RoboDK station: ur3.rdk

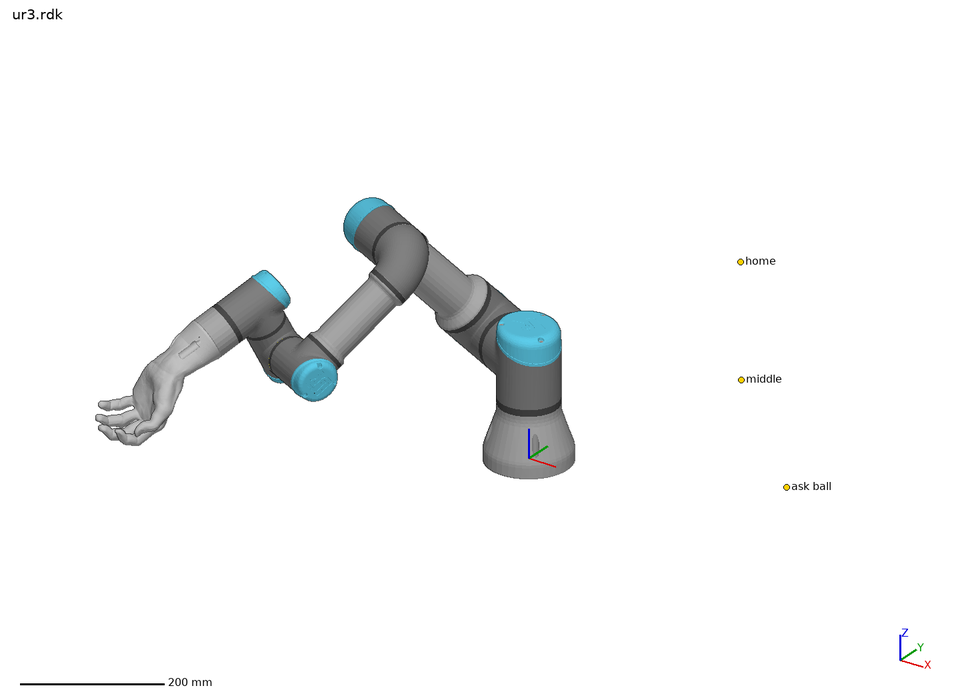
[picture v0: the station drawn from its stored meshes, robots at their saved joint values, targets as dots, program paths as lines]
Station ur3 (saved by RoboDK 5.9.2). Poses are relative to the parent item; angles as X-Y-Z fixed-axis rotations.
  - frame UR3 Base at (0, 0, 0) mm
    - robot UR3: 6 axes, payload 3 kg, reach 500 mm, repeatability 0.1 mm, weight 11 kg
        modified DH rows (alpha deg, a mm, theta deg, d mm): 0, 0, 0, 151.9; 90, 0, 180, 0; 0, 243.65, 0, 0; 0, 213, 0, 110.4; -90, 0, 0, 83.4; 90, 0, 180, 82.4
        joint limits [-360, -360, -360, -360, -360, -360] to [360, 360, 360, 360, 360, 360]; home [0, -90, -90, 0, 90, 0]; saved at [-117.843, -133.139, -84.851, 11.276, 90.861, -184.017]
      - tool hand_ballholding_02, TCP at (0, 10, 140) mm, size 105.6 x 100.7 x 194.6 mm, geometry from hand_ballholding_02.stl
    - target home (Cartesian target) at (435.4, -110.28, 468.95) mm, rotated rx -90 ry 0.68 rz -90 deg; joints [0, -90, -90, 0, 90, 0.68] of UR3
    - target middle (Cartesian target) at (435.4, -108.11, 285.91) mm, rotated rx -90 ry 0.68 rz -90 deg; joints [0.586, -109.669, -122.761, 52.43, 89.414, 0.68] of UR3
    - target ask ball (Cartesian target) at (510.58, -106.39, 140.74) mm, rotated rx -113.61 ry 0.68 rz -90 deg; joints [0.526, -129.977, -105.78, 32.153, 89.79, 0.834] of UR3
  - Python program Prog1 (listed below)

--- Python program Prog1 ---
from robodk import robolink, robomath
from pythonosc import dispatcher, osc_server
from pythonosc.osc_server import ThreadingOSCUDPServer
import math

# Connect to RoboDK
RDK = robolink.Robolink()
robot = RDK.Item('UR3e')  # change to your robot name in RoboDK

def deg_to_rad(deg):
    return deg * math.pi / 180.0

# MoveJ handler (RoboDK version of your ur_rtde handler)
def handle_movej(unused_addr, *args):
    if len(args) not in [6, 8]:
        print("Expected 6 joint values (°), optionally followed by acceleration and joint speed.")
        return
    try:
        joint_positions = list(args[:6])

        # Default defaults
        accel = 100.0  # deg/s²
        speed = 30.0   # deg/s

        if len(args) == 8:
            accel = args[7] / 5
            speed = args[6] / 5

        # Correct methods from RoboDK API:
        robot.setAccelerationJoints(accel)
        robot.setSpeedJoints(speed)
        print(f"Joint accel set to {accel} deg/s², speed set to {speed} deg/s")

        robot.MoveJ(joint_positions)
        print(f"RoboDK MoveJ executed: {joint_positions} (°)")

    except Exception as e:
        print(f"RoboDK MoveJ error: {e}")


import time
import threading

latest_target = None
target_lock = threading.Lock()

# OSC handler just stores the latest target
def handle_servoj(unused_addr, *args):
    global latest_target
    if len(args) < 6:
        return
    with target_lock:
        latest_target = list(args[:6])  # store latest joint target

# Worker thread updates robot at fixed rate
def servoj_worker():
    global latest_target
    update_rate = 0.03  # 10 Hz (0.1s)
    robot.setSpeedJoints(1000)
    robot.setAccelerationJoints(1000)
    while True:
        target = None
        with target_lock:
            if latest_target is not None:
                target = latest_target
                latest_target = None  # clear after taking it
        if target:
            robot.MoveJ(target)
            print(f"RoboDK servoj executed: {target}")
        time.sleep(update_rate)

# Start the worker in a separate thread
threading.Thread(target=servoj_worker, daemon=True).start()


# MoveL handler (same idea)
def handle_movel(unused_addr, *args):
    if len(args) not in [6, 8]:
        print("Expected 6 pose values (x, y, z in m, rx, ry, rz in °), optionally followed by accel/speed.")
        return
    try:
        pose = list(args[:3]) + [deg_to_rad(val) for val in args[3:6]]
        robot.MoveL(pose)
        print(f"RoboDK MoveL executed: {pose}")
    except Exception as e:
        print(f"RoboDK MoveL error: {e}")

# Setup OSC dispatcher
dispatcher = dispatcher.Dispatcher()
dispatcher.map("/movej", handle_movej)
dispatcher.map("/movel", handle_movel)
dispatcher.map("/servoj", handle_servoj)

# OSC server
OSC_LISTEN_IP = "0.0.0.0"
OSC_LISTEN_PORT = 9001
server = ThreadingOSCUDPServer((OSC_LISTEN_IP, OSC_LISTEN_PORT), dispatcher)
print(f"RoboDK listening for OSC on {OSC_LISTEN_IP}:{OSC_LISTEN_PORT}")

server.serve_forever()
